SYSTEM test
  (* Standard: 61499-1; Classification: Training; ApplicationDomain: Agriculture; Function: Learning how to use 4diac; Type: Test Type; Description: Copyright (c) 2023 HR Agrartechnik GmbH This program and the accompanying materials are made available under the terms of the Eclipse Public License 2.0 which is available at https://www.eclipse.org/legal/epl-2.0/ SPDX-License-Identifier: EPL-2.0 Training Hier kann man über "Change Type" andere Ventilsteuerung_Uebung_001 usw auswählen, und so Übung für Übung vollziehen. Quellen: 1. Mit Musterlösungen: https://github.com/Meisterschulen-am-Ostbahnhof-Munchen/4diac_training1 2. Ohne Musterlösungen: https://github.com/Meisterschulen-am-Ostbahnhof-Munchen/4diac_training1_empty *)
  (* Version 1.0, 2023-10-23, Franz Höpfinger, HR Agrartechnik GmbH *)
  PACKAGE Training;
  IMPORT logiBUS::stations::Computers::C_ST;
  APPLICATION App (* Default App for Everything *)
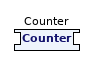
    SUBAPPS
      Counter : Counter;
    END_SUBAPPS
  END_APPLICATION
  DEVICE FORTE_PC : iec61499::system::FORTE_PC(MGR_ID := C_ST (* Device manager socket ID *))
    {SET_ATTRIBUTE(Profile, HOLOBLOC)}
    RESOURCE EMB_RES : iec61499::system::EMB_RES
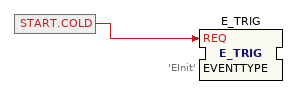
      FBS
        E_TRIG : iec61499::events::E_TRIG(EVENTTYPE := 'EInit');
      END_FBS
      EVENT_CONNECTIONS
        START.COLD TO E_TRIG.REQ;
      END_CONNECTIONS
    END_RESOURCE
  END_DEVICE
  MAPPINGS
    App.Counter ON FORTE_PC.EMB_RES;
  END_MAPPINGS
  SEGMENTS
    Ethernet : iec61499::system::Ethernet;
  END_SEGMENTS
  LINKS
    FORTE_PC => Ethernet;
  END_LINKS
END_SYSTEM
